// TwinCAT 3 PLC project TcoInspectorsTests
// Title: TcoInspectorsTests
// Company: Vortex.Library
// ProjectVersion: 0.6.0.913
// ProgramVersion: 3.1.4024.12
// libraries:
//   Tc2_Standard, * (Beckhoff Automation GmbH)
//   Tc2_System, * (Beckhoff Automation GmbH)
//   Tc3_Module, * (Beckhoff Automation GmbH)
//   TcoCore, 0.6.0.913 (Vortex.Library)
//   TcoInspectors, 0.6.0.913 (Vortex.Library)
// project tree:
//   GVLs/ GVL.TcGVL
//   / PlcTask.TcTTO
//   POUs/Examples/ ExampleComponents.TcDUT, ExampleContext.TcPOU, ExampleDimensionsInspectors.TcDUT, ExampleInspectorsStruct.TcDUT, Examples_2.TcPOU, ExamplesImplementationWithDone.TcPOU, Sequence1Task.TcPOU
//   POUs/ MAIN.TcPOU
//   POUs/Mocks/ MockCoordinator.TcPOU
//   POUs/Tests/TcoAnalogueInspector/ TcoAnalogueInspectorTests.TcPOU
//   POUs/Tests/TcoDataInspector/ TcoDataInspectorTests.TcPOU
//   POUs/Tests/TcoDigitalInspector/Legacy/ eDigitalInspectorTests.TcDUT, LegacyTcoDigitalInspectorTests.TcPOU
//   POUs/Tests/TcoDigitalInspector/ TcoDigitalInspectorTests.TcPOU
//   POUs/Tests/TcoInspectionGroup/ eInspectionGroupTests.TcDUT, TcoInspectionGroupTests.TcPOU
//   POUs/Tests/TcoInspector/ eInspectorTests.TcDUT, TcoInspectorTests.TcPOU
// (motion and I/O tree: see PLC project tcoinspectors)
// real-time tasks:
//   TASK PlcTask: cycle T#10ms, priority 20, ADS port 350
//   TASK PlcTask1: cycle T#10ms, priority 21, ADS port 351

CONFIGURATION TcoInspectorsTests
    RESOURCE PLC ON TwinCAT3
        TASK PlcTask(INTERVAL := T#10ms, PRIORITY := 21);
        PROGRAM MAIN WITH PlcTask : MAIN;
    END_RESOURCE
END_CONFIGURATION

// ---- POUs/Examples/ExampleComponents.TcDUT
TYPE ExampleComponents EXTENDS TcoCore.TcoStruct :
STRUCT
    DmcReader : STRING;
    BoltPresenceSensor : BOOL;
    DimX_Sensor : LREAL;
    DimY_Sensor : LREAL;
    DimZ_Sensor : LREAL;
END_STRUCT
END_TYPE

// ---- POUs/Examples/ExampleDimensionsInspectors.TcDUT
TYPE ExampleDimensionsInspectors EXTENDS TcoCore.TcoStruct :
STRUCT
    {attribute addProperty Name "Dimension X inspection"}
    DimX_Inspector : TcoInspectors.TcoAnalogueInspector(THISSTRUCT);
    {attribute addProperty Name "Dimension Y inspection"}
    DimY_Inspector : TcoInspectors.TcoAnalogueInspector(THISSTRUCT);
    {attribute addProperty Name "Dimension ZZ inspection"}
    DimZ_Inspector : TcoInspectors.TcoAnalogueInspector(THISSTRUCT);
    {attribute addProperty Name "Dimension Z inspection name is TOOOOOOOO LONG"}
    DimCustom_Inspector : TcoInspectors.TcoAnalogueInspector(THISSTRUCT);
    {attribute addProperty Name "Dimension inspection 1"}
    Dim_Inspector_1 : TcoInspectors.TcoAnalogueInspector(THISSTRUCT);
    {attribute addProperty Name "Dimension inspection 2"}
    Dim_Inspector_2 : TcoInspectors.TcoAnalogueInspector(THISSTRUCT);
    {attribute addProperty Name "Dimension inspection 3"}
    Dim_Inspector_3 : TcoInspectors.TcoAnalogueInspector(THISSTRUCT);
    {attribute addProperty Name "Dimension inspection 4"}
    Dim_Inspector_4 : TcoInspectors.TcoAnalogueInspector(THISSTRUCT);
    {attribute addProperty Name "Dimension inspection 5"}
    Dim_Inspector_5 : TcoInspectors.TcoAnalogueInspector(THISSTRUCT);
    {attribute addProperty Name "Dimension inspection 6"}
    Dim_Inspector_6 : TcoInspectors.TcoAnalogueInspector(THISSTRUCT);
    {attribute addProperty Name "Dimension inspection 7"}
    Dim_Inspector_7 : TcoInspectors.TcoAnalogueInspector(THISSTRUCT);
    {attribute addProperty Name "Dimension inspection 8"}
    Dim_Inspector_8 : TcoInspectors.TcoAnalogueInspector(THISSTRUCT);
    {attribute addProperty Name "Dimension inspection 9"}
    Dim_Inspector_9 : TcoInspectors.TcoAnalogueInspector(THISSTRUCT);
    {attribute addProperty Name "Dimension inspection 10"}
    Dim_Inspector_10 : TcoInspectors.TcoAnalogueInspector(THISSTRUCT);
    {attribute addProperty Name "Dimension inspection 11"}
    Dim_Inspector_11 : TcoInspectors.TcoAnalogueInspector(THISSTRUCT);
    {attribute addProperty Name "Dimension inspection 12"}
    Dim_Inspector_12 : TcoInspectors.TcoAnalogueInspector(THISSTRUCT);
    {attribute addProperty Name "Dimension inspection 13"}
    Dim_Inspector_13 : TcoInspectors.TcoAnalogueInspector(THISSTRUCT);
    {attribute addProperty Name "Dimension inspection 14"}
    Dim_Inspector_14 : TcoInspectors.TcoAnalogueInspector(THISSTRUCT);
    {attribute addProperty Name "Dimension inspection 15"}
    Dim_Inspector_15 : TcoInspectors.TcoAnalogueInspector(THISSTRUCT);
    {attribute addProperty Name "Dimension inspection 16"}
    Dim_Inspector_16 : TcoInspectors.TcoAnalogueInspector(THISSTRUCT);
    {attribute addProperty Name "Dimension inspection 17"}
    Dim_Inspector_17 : TcoInspectors.TcoAnalogueInspector(THISSTRUCT);
    {attribute addProperty Name "Dimension inspection 18"}
    Dim_Inspector_18 : TcoInspectors.TcoAnalogueInspector(THISSTRUCT);
    {attribute addProperty Name "Dimension inspection 19"}
    Dim_Inspector_19 : TcoInspectors.TcoAnalogueInspector(THISSTRUCT);
    {attribute addProperty Name "Dimension inspection 20"}
    Dim_Inspector_20 : TcoInspectors.TcoAnalogueInspector(THISSTRUCT);
//Inspectors : ARRAY[0..20] OF TcoInspectors.TcoAnalogueInspector(THISSTRUCT);
END_STRUCT
END_TYPE

// ---- POUs/Examples/ExampleInspectorsStruct.TcDUT
TYPE ExampleInspectorsStruct EXTENDS TcoCore.TcoStruct :
STRUCT
    {attribute addProperty Name "Overall result"}
    OverallResult : TcoInspectors.TcoComprehensiveResult;
    {attribute addProperty Name "DMC code inspection"}
    DmcInspector : TcoInspectors.TcoDataInspector(THISSTRUCT);
    {attribute addProperty Name "Bolt presence inspection"}
    BoltPresenceInspector : TcoInspectors.TcoDigitalInspector(THISSTRUCT);
    Dimensions : ExampleDimensionsInspectors := (Parent := THISSTRUCT);
END_STRUCT
END_TYPE

// ---- POUs/Tests/TcoDigitalInspector/Legacy/eDigitalInspectorTests.TcDUT
{attribute 'qualified_only'}
{attribute 'strict'}
TYPE eDigitalInspectorTests :
(
    Inspect := 10,
    GetResult := 20,
    UpdateOverall := 30,
    OnFailCarryOn := 40,
    OnFailRetry := 50,
    OnFailTerminate := 60
);
END_TYPE

// ---- POUs/Tests/TcoInspectionGroup/eInspectionGroupTests.TcDUT
{attribute 'qualified_only'}
{attribute 'strict'}
TYPE eInspectionGroupTests :
(
    Inspect := 10,
    GetResult := 20,
    OnFailCarryOn := 40,
    OnFailRetry := 50,
    OnFailTerminate := 60,
    OnFailDiaglog := 70,
    InspectWithNormalizedNumberOfRetries := 80,
    UpdateComprehensiveResultDescriptions := 90
);
END_TYPE

// ---- POUs/Tests/TcoInspector/eInspectorTests.TcDUT
{attribute 'qualified_only'}
{attribute 'strict'}
TYPE eInspectorTests :
(
    Inspect := 10,
    GetResult := 20,
    UpdateOverall := 30,
    OnFailCarryOn := 40,
    OnFailRetry := 50,
    OnFailTerminate := 60,
    OnFailDialog := 70
);
END_TYPE

// ---- GVLs/GVL.TcGVL
{attribute 'qualified_only'}
VAR_GLOBAL
END_VAR

// ---- POUs/MAIN.TcPOU
PROGRAM MAIN
VAR
    _legacyDigitalInspectorTests : LegacyTcoDigitalInspectorTests;
    _digitalInspectorTests : TcoDigitalInspectorTests;
    _analogueInspectorTests : TcoAnalogueInspectorTests;
    _dataInspectorTests : TcoDataInspectorTests;
    _inspectionGroupTests : TcoInspectionGroupTests;
    _exampleContext : ExampleContext;
END_VAR

_legacyDigitalInspectorTests.ProbeRun();
_digitalInspectorTests.ProbeRun();
_analogueInspectorTests.ProbeRun();
_dataInspectorTests.ProbeRun();
_inspectionGroupTests.ProbeRun();
_exampleContext.Run();

END_PROGRAM

// ---- POUs/Tests/TcoDigitalInspector/Legacy/LegacyTcoDigitalInspectorTests.TcPOU
FUNCTION_BLOCK LegacyTcoDigitalInspectorTests EXTENDS TcoCore._internals_TcoContext
VAR
    _sut : TcoInspectors.TcoDigitalInspector(THIS^);
    _inspectedValue : BOOL;
    _result : TcoInspectors.eInspectorResult;
    _isOverIspected : BOOL;
    _overallResult : TcoInspectors.TcoComprehensiveResult;
    _coordinator : MockCoordinator;
    i_coordinator : TcoCore.ITcoCoordinator;
    _retryState : INT;
END_VAR

METHOD PROTECTED Main
i_coordinator := _coordinator;

CASE _testId OF
    0:
        _result := 0;
        _isOverIspected := FALSE;
    eDigitalInspectorTests.Inspect:
        THIS^.ProbeDoneWhen(_sut.Inspect(_inspectedValue).UpdateComprehensiveResult(_overallResult).Done);
    eDigitalInspectorTests.GetResult:
        _result := _sut.Inspect(_inspectedValue).Result;
        _isOverIspected := _sut.Inspect(_inspectedValue).OverInspected;
    eDigitalInspectorTests.OnFailCarryOn:
        THIS^.ProbeDoneWhen(_sut.WithCoordinator(i_coordinator).Inspect(_inspectedValue).OnFail().CarryOn());
    eDigitalInspectorTests.OnFailRetry:
        THIS^.ProbeDoneWhen(_sut.WithCoordinator(i_coordinator).Inspect(_inspectedValue).OnFail().Retry(_retryState));
    eDigitalInspectorTests.OnFailTerminate:
        THIS^.ProbeDoneWhen(_sut.WithCoordinator(i_coordinator).Inspect(_inspectedValue).OnFail().Terminate());
END_CASE
END_METHOD

END_FUNCTION_BLOCK

// ---- POUs/Mocks/MockCoordinator.TcPOU
FUNCTION_BLOCK MockCoordinator IMPLEMENTS TcoCore.ITcoCoordinator
VAR
    _state : INT;
END_VAR

PROPERTY IsFreshState : BOOL
GET
END_GET
END_PROPERTY

METHOD MoveNext : BOOL
_state := _state + 1;
END_METHOD

METHOD Retry : BOOL
VAR_INPUT
    inFromState : INT;
END_VAR
_state := inFromState;
END_METHOD

METHOD Terminate : BOOL
_state := 8005;
END_METHOD

END_FUNCTION_BLOCK

// ---- POUs/Tests/TcoDigitalInspector/TcoDigitalInspectorTests.TcPOU
FUNCTION_BLOCK TcoDigitalInspectorTests EXTENDS TcoInspectorTests
VAR
    _sut : TcoInspectors.TcoDigitalInspector(THIS^);
    _inspectedValue : BOOL;
END_VAR

METHOD Inspect : TcoInspectors.IInspector
Inspect := _sut.Inspect(_inspectedValue);
END_METHOD

METHOD PROTECTED Main
SUPER^.Main();
END_METHOD

METHOD WithCoordinator : REFERENCE TO TcoInspectorTests
VAR_INPUT
    inoCoordinator : TcoCore.ITcoCoordinator;
END_VAR
_sut.WithCoordinator(_coordinator);
WithCoordinator REF= THIS^;
END_METHOD

END_FUNCTION_BLOCK

// ---- POUs/Tests/TcoInspector/TcoInspectorTests.TcPOU
FUNCTION_BLOCK ABSTRACT TcoInspectorTests EXTENDS TcoCore._internals_TcoContext
VAR
    _result : TcoInspectors.eInspectorResult;
    _isOverIspected : BOOL;
    _overallResult : TcoInspectors.TcoComprehensiveResult;
    _coordinator : MockCoordinator;
    i_coordinator : TcoCore.ITcoCoordinator;
    _retryState : INT;
END_VAR

METHOD ABSTRACT Inspect : TcoInspectors.IInspector
END_METHOD

METHOD PROTECTED Main
i_coordinator := _coordinator;

CASE _testId OF
    0:
        _result := 0;
        _isOverIspected := FALSE;
    eInspectorTests.Inspect:
        THIS^.ProbeDoneWhen(Inspect().UpdateComprehensiveResult(_overallResult).Done);
    eInspectorTests.GetResult:
        _result := Inspect().Result;
        _isOverIspected := Inspect().OverInspected;
    eInspectorTests.OnFailCarryOn:
        THIS^.ProbeDoneWhen(WithCoordinator(inoCoordinator := i_coordinator).Inspect().OnFail().CarryOn());
    eInspectorTests.OnFailRetry:
        THIS^.ProbeDoneWhen(WithCoordinator(inoCoordinator := i_coordinator).Inspect().OnFail().Retry(_retryState));
    eInspectorTests.OnFailTerminate:
        THIS^.ProbeDoneWhen(WithCoordinator(inoCoordinator := i_coordinator).Inspect().OnFail().Terminate());
    eInspectorTests.OnFailDialog:
        THIS^.ProbeDoneWhen(WithCoordinator(inoCoordinator := i_coordinator).Inspect().OnFail().Dialog(100));
END_CASE
END_METHOD

METHOD ABSTRACT WithCoordinator : REFERENCE TO TcoInspectorTests
VAR_INPUT
    inoCoordinator : TcoCore.ITcoCoordinator;
END_VAR
END_METHOD

END_FUNCTION_BLOCK

// ---- POUs/Tests/TcoAnalogueInspector/TcoAnalogueInspectorTests.TcPOU
FUNCTION_BLOCK TcoAnalogueInspectorTests EXTENDS TcoInspectorTests
VAR
    _sut : TcoInspectors.TcoAnalogueInspector(THIS^);
    _inspectedValue : LREAL;
END_VAR

METHOD Inspect : TcoInspectors.IInspector
Inspect := _sut.Inspect(_inspectedValue);
END_METHOD

METHOD PROTECTED Main
SUPER^.Main();
END_METHOD

METHOD WithCoordinator : REFERENCE TO TcoInspectorTests
VAR_INPUT
    inoCoordinator : TcoCore.ITcoCoordinator;
END_VAR
_sut.WithCoordinator(_coordinator);
WithCoordinator REF= THIS^;
END_METHOD

END_FUNCTION_BLOCK

// ---- POUs/Tests/TcoDataInspector/TcoDataInspectorTests.TcPOU
FUNCTION_BLOCK TcoDataInspectorTests EXTENDS TcoInspectorTests
VAR
    _sut : TcoInspectors.TcoDataInspector(THIS^);
    _inspectedValue : STRING;
END_VAR

METHOD Inspect : TcoInspectors.IInspector
Inspect := _sut.Inspect(_inspectedValue);
END_METHOD

METHOD PROTECTED Main
SUPER^.Main();
END_METHOD

METHOD WithCoordinator : REFERENCE TO TcoInspectorTests
VAR_INPUT
    inoCoordinator : TcoCore.ITcoCoordinator;
END_VAR
_sut.WithCoordinator(_coordinator);
WithCoordinator REF= THIS^;
END_METHOD

END_FUNCTION_BLOCK

// ---- POUs/Tests/TcoInspectionGroup/TcoInspectionGroupTests.TcPOU
FUNCTION_BLOCK TcoInspectionGroupTests EXTENDS TcoCore._internals_TcoContext
VAR
    _sut : TcoInspectors.TcoInspectionGroup(THIS^);
    _diis : ARRAY[0..1] OF TcoInspectors.TcoDigitalInspector(THIS^);
    _dii_inspectedValues : ARRAY[0..1] OF BOOL;
    _dais : ARRAY[0..1] OF TcoInspectors.TcoAnalogueInspector(THIS^);
    _dai_inspectedValues : ARRAY[0..1] OF REAL;
    _ddis : ARRAY[0..1] OF TcoInspectors.TcoDataInspector(THIS^);
    _ddi_inspectedValues : ARRAY[0..1] OF STRING;
    _overallResult : TcoInspectors.TcoComprehensiveResult;
    _coordinator : MockCoordinator;
    _retryState : INT;
    _tmp : ITcoInspectionGroupAct;
END_VAR

METHOD PROTECTED Main
CASE _testId OF
    eInspectionGroupTests.Inspect:
        THIS^.ProbeDoneWhen(_sut.Act()
                .Inspect(_diis[0].Inspect(_dii_inspectedValues[0]))
                .Inspect(_diis[1].Inspect(_dii_inspectedValues[1]))
                .Inspect(_dais[0].Inspect(_dai_inspectedValues[0]))
                .Inspect(_dais[1].Inspect(_dai_inspectedValues[1]))
                .Inspect(_ddis[0].Inspect(_ddi_inspectedValues[0]))
                .Inspect(_ddis[1].Inspect(_ddi_inspectedValues[1]))
                .UpdateComprehensiveResult(_overallResult).Done);
    eInspectionGroupTests.OnFailCarryOn:
        THIS^.ProbeDoneWhen(_sut.WithCoordinator(_coordinator)
                .Act()
                .Inspect(_diis[0].Inspect(_dii_inspectedValues[0]))
                .Inspect(_diis[1].Inspect(_dii_inspectedValues[1]))
                .Inspect(_dais[0].Inspect(_dai_inspectedValues[0]))
                .Inspect(_dais[1].Inspect(_dai_inspectedValues[1]))
                .Inspect(_ddis[0].Inspect(_ddi_inspectedValues[0]))
                .Inspect(_ddis[1].Inspect(_ddi_inspectedValues[1]))
                .UpdateComprehensiveResult(_overallResult)
                .OnFail()
                .CarryOn());
    eInspectionGroupTests.OnFailRetry:
        THIS^.ProbeDoneWhen(_sut.WithCoordinator(_coordinator)
                .Act()
                .Inspect(_diis[0].Inspect(_dii_inspectedValues[0]))
                .Inspect(_diis[1].Inspect(_dii_inspectedValues[1]))
                .Inspect(_dais[0].Inspect(_dai_inspectedValues[0]))
                .Inspect(_dais[1].Inspect(_dai_inspectedValues[1]))
                .Inspect(_ddis[0].Inspect(_ddi_inspectedValues[0]))
                .Inspect(_ddis[1].Inspect(_ddi_inspectedValues[1]))
                .UpdateComprehensiveResult(_overallResult)
                .OnFail()
                .Retry(_retryState));
    eInspectionGroupTests.OnFailTerminate:
        THIS^.ProbeDoneWhen(_sut.WithCoordinator(_coordinator)
                .Act()
                .Inspect(_diis[0].Inspect(_dii_inspectedValues[0]))
                .Inspect(_diis[1].Inspect(_dii_inspectedValues[1]))
                .Inspect(_dais[0].Inspect(_dai_inspectedValues[0]))
                .Inspect(_dais[1].Inspect(_dai_inspectedValues[1]))
                .Inspect(_ddis[0].Inspect(_ddi_inspectedValues[0]))
                .Inspect(_ddis[1].Inspect(_ddi_inspectedValues[1]))
                .UpdateComprehensiveResult(_overallResult)
                .OnFail()
                .Terminate());
    eInspectionGroupTests.OnFailDiaglog:
        THIS^.ProbeDoneWhen(_sut.WithCoordinator(_coordinator)
                .Act()
                .Inspect(_diis[0].Inspect(_dii_inspectedValues[0]))
                .Inspect(_diis[1].Inspect(_dii_inspectedValues[1]))
                .Inspect(_dais[0].Inspect(_dai_inspectedValues[0]))
                .Inspect(_dais[1].Inspect(_dai_inspectedValues[1]))
                .Inspect(_ddis[0].Inspect(_ddi_inspectedValues[0]))
                .Inspect(_ddis[1].Inspect(_ddi_inspectedValues[1]))
                .UpdateComprehensiveResult(_overallResult)
                .OnFail()
                .Dialog(100));
    eInspectionGroupTests.InspectWithNormalizedNumberOfRetries:
        THIS^.ProbeDoneWhen(_sut.WithCoordinator(_coordinator)
                .Act()
                .NormalizeRetries(_diis[0])
                .NormalizeRetries(_diis[1])
                .NormalizeRetries(_dais[0])
                .NormalizeRetries(_dais[1])
                .NormalizeRetries(_ddis[0])
                .NormalizeRetries(_ddis[1])
                .Inspect(_diis[0].Inspect(_dii_inspectedValues[0]))
                .Inspect(_diis[1].Inspect(_dii_inspectedValues[1]))
                .Inspect(_dais[0].Inspect(_dai_inspectedValues[0]))
                .Inspect(_dais[1].Inspect(_dai_inspectedValues[1]))
                .Inspect(_ddis[0].Inspect(_ddi_inspectedValues[0]))
                .Inspect(_ddis[1].Inspect(_ddi_inspectedValues[1]))
                .UpdateComprehensiveResult(_overallResult).Done);
    eInspectionGroupTests.UpdateComprehensiveResultDescriptions:
        THIS^.ProbeDoneWhen(_sut.WithCoordinator(_coordinator)
                .Act()
                .NormalizeRetries(_diis[0])
                .NormalizeRetries(_diis[1])
                .NormalizeRetries(_dais[0])
                .NormalizeRetries(_dais[1])
                .NormalizeRetries(_ddis[0])
                .NormalizeRetries(_ddis[1])
                .Inspect(_diis[0].Inspect(_dii_inspectedValues[0]))
                .Inspect(_diis[1].Inspect(_dii_inspectedValues[1]))
                .Inspect(_dais[0].Inspect(_dai_inspectedValues[0]))
                .Inspect(_dais[1].Inspect(_dai_inspectedValues[1]))
                .Inspect(_ddis[0].Inspect(_ddi_inspectedValues[0]))
                .Inspect(_ddis[1].Inspect(_ddi_inspectedValues[1]))
                .UpdateComprehensiveResult(_overallResult)
                .OnFail()
                .Dialog(100));
END_CASE
END_METHOD

END_FUNCTION_BLOCK

// ---- POUs/Examples/ExampleContext.TcPOU
FUNCTION_BLOCK ExampleContext EXTENDS TcoCore.TcoContext
VAR
    Data            : ExampleInspectorsStruct := (Parent := THIS^);
    Components      : ExampleComponents       := (Parent := THIS^);
    GroupInspection : TcoInspectors.TcoInspectionGroup(THIS^);
    _sequence1      : TcoCore.TcoSequence(THIS^, eRestoreMode.None);
    _observer       : TcoCore.TcoSequencerObserver(THIS^);
    {attribute addProperty Name "Start sequence"}
    _sequence1Task 	: Sequence1Task(THIS^);
    _dialog        	: TcoCore.TcoDialog(THIS^);
    {attribute 'hide'}
    EmptyData 		: ExampleInspectorsStruct := (Parent := THIS^);

    _examples_2 	: Examples_2(THIS^);
	_examplesImplementationWithDone : ExamplesImplementationWithDone(THIS^);
	_tonRetry: TON;
	_rtrigRetry: R_trig;
	_tonTerminate: TON;
	testRetry:BOOL;
	testTerminate:BOOL;
	
END_VAR

(*~
	<docu>
		<summary>
			Main method of the TcoContext. This is the entry point of any control logic that belongs to this context. 
			The call of this method is ensured by calling the <c>InstanceName.Run()</c> method, and it must not be called explicitly.
			This method is abstract, and it must be overridden in derived block.
		</summary>
	</docu>
~*)
METHOD PROTECTED  Main
_sequence1Task(Sequence := _sequence1);
IF(_sequence1Task.Execute())THEN
	Sequence1();
END_IF;

_examples_2();
_examplesImplementationWithDone();
END_METHOD

METHOD Sequence1
VAR
    seq    : REFERENCE TO TcoCore.TcoSequence;
    answer : TcoCore.eDialogAnswer;
	i: INT;
END_VAR
seq REF= _sequence1;

seq.Open();
seq.Observer := _observer;

IF (seq.Step(inStepID := 0,
    inEnabled := TRUE,
    inStepDescription := 'ASKING SOME QUESTION')) THEN
    //--------------------------------------------------------
    //<StandardDialog>	
    //restore method also close inactive dialog
    Data.BoltPresenceInspector.Restore();
    GroupInspection.Restore();
    SetupData();
    answer := _dialog
        .Show()
        .WithType(eDialogType.Question)
        .WithCaption('Ready to go?')
        .WithText('We are about to start the inspection sequence. Do we go ahead?')
        .WithYesNoCancel().Answer;

    //

    IF (answer = TcoCore.eDialogAnswer.Yes) THEN
        seq.CompleteStep();
    ELSIF (answer = TcoCore.eDialogAnswer.No) THEN
        _sequence1Task.Restore();
    ELSIF (answer = TcoCore.eDialogAnswer.Cancel) THEN
        seq.RequestStep(400);
    END_IF;
    //</StandardDialog>	 
    //--------------------------------------------------------			
END_IF;

IF (seq.Step(inStepID := 25,
    inEnabled := TRUE,
    inStepDescription := 'SETUP DATA')) THEN
    //--------------------------------------------------------    
    SetupData();
    seq.CompleteStep();
    //--------------------------------------------------------			
END_IF;

IF (seq.Step(inStepID := 50,
    inEnabled := TRUE,
    inStepDescription := 'INIT')) THEN
    //--------------------------------------------------------    	 	       
    seq.CompleteStep();
    //--------------------------------------------------------			
END_IF;

IF (seq.Step(inStepID := 100,
    inEnabled := TRUE,
    inStepDescription := 'INSPECT DMC CODE - WHEN CARRY ON')) THEN
    //--------------------------------------------------------
    Data.DmcInspector.WithCoordinator(seq)
        .Inspect(Components.DmcReader)
        .UpdateComprehensiveResult(Data.OverallResult)
        .OnFail()
        .CarryOn();
    //--------------------------------------------------------			
END_IF;

IF (seq.Step(inStepID := 105,
    inEnabled := TRUE,
    inStepDescription := 'SETUP DATA')) THEN
    //--------------------------------------------------------    
    SetupData();
    seq.CompleteStep();
    //--------------------------------------------------------			
END_IF;

IF (seq.Step(inStepID := 110,
    inEnabled := TRUE,
    inStepDescription := 'DUMMY WAIT')) THEN
    //--------------------------------------------------------
    seq.StepCompleteWhen(Seq.CurrentStep.Duration > T#1S);
    //--------------------------------------------------------			
END_IF;

IF (seq.Step(inStepID := 120,
    inEnabled := TRUE,
    inStepDescription := 'INSPECT DMC CODE -  RETRY THEN TERMINATE')) THEN
    //--------------------------------------------------------
    Data.DmcInspector.WithCoordinator(seq)
        .Inspect(Components.DmcReader)
        .UpdateComprehensiveResult(Data.OverallResult)
        .OnFail()
        .RetryThenTerminate(110);
    //--------------------------------------------------------			
END_IF;

//<TcoDigitalInspector>	
IF (seq.Step(inStepID := 200,
    inEnabled := true,
    inStepDescription := 'INSPECT BOLT PRESENCE - ASK WHAT TO DO')) THEN
    //--------------------------------------------------------	
    IF seq.IsFreshState THEN
        SetupData();
    END_IF

    Data.BoltPresenceInspector
        .WithCoordinator(seq)
        .Inspect(Components.BoltPresenceSensor)
        .UpdateComprehensiveResult(Data.OverallResult)
        .OnFail()
        .Dialog(seq.CurrentStep.ID + 1);
    //--------------------------------------------------------			
END_IF;

IF (seq.Step(inStepID := 201,
    inEnabled := true,
    inStepDescription := 'INSPECT BOLT PRESENCE - ASK WHAT TO DO WITH INSTRUCTION')) THEN
    //--------------------------------------------------------	
    IF seq.IsFreshState THEN
        SetupData();
    END_IF

    Data.BoltPresenceInspector
        .WithCoordinator(seq)
        .Inspect(Components.BoltPresenceSensor)
        .UpdateComprehensiveResult(Data.OverallResult)
        .Instruct('Something is wrong')
        .OnFail()
        .Dialog(seq.CurrentStep.ID + 1);
    //--------------------------------------------------------			
END_IF;

IF (seq.Step(inStepID := 202,
    inEnabled := true,
    inStepDescription := 'INSPECT BOLT PRESENCE - ASK WHAT TO DO WITH INSTRUCTION AND PICTURE')) THEN
    //--------------------------------------------------------	
    IF seq.IsFreshState THEN
        SetupData();
    END_IF

    Data.BoltPresenceInspector
        .WithCoordinator(seq)
        .Inspect(Components.BoltPresenceSensor)
        .UpdateComprehensiveResult(Data.OverallResult)
        .Instruct('Something is wrong')
        .InstructWithImage('d:\MTS\Develop\TcOpenGroup\TcOpen\assets\logo\TcOpenWide.png', 200, 200)
        .OnFail()
        .Dialog(seq.CurrentStep.ID + 1);
    //--------------------------------------------------------			
END_IF;

IF (seq.Step(inStepID := 203,
    inEnabled := true,
    inStepDescription := 'INSPECT BOLT PRESENCE - ASK WHAT TO DO WITH INSTRUCTION AND BIGGER PICTURE')) THEN
    //--------------------------------------------------------	
    IF seq.IsFreshState THEN
        SetupData();
    END_IF

    Data.BoltPresenceInspector
        .WithCoordinator(seq)
        .Inspect(Components.BoltPresenceSensor)
        .UpdateComprehensiveResult(Data.OverallResult)
        .Instruct('Something is wrong') //provide cuastomized instruction instead of automaticaly generated
        .InstructWithImage('d:\MTS\Develop\TcOpenGroup\TcOpen\assets\logo\TcOpenWide.png', 600, 600)
        .OnFail()
        .Dialog(seq.CurrentStep.ID + 1);
    //--------------------------------------------------------			
END_IF;

IF (seq.Step(inStepID := 204,
    inEnabled := true,
    inStepDescription := 'INSPECT BOLT PRESENCE - ASK WHAT TO DO WITH FAILURE DESCRIPTION')) THEN
    //--------------------------------------------------------	
    IF seq.IsFreshState THEN
        SetupData();
    END_IF

    Data.BoltPresenceInspector
        .WithCoordinator(seq)
        .Inspect(Components.BoltPresenceSensor)
        .UpdateComprehensiveResult(Data.OverallResult)
        .WithFailureDescription()
        .OnFail()
        .Dialog(seq.CurrentStep.ID + 1);
    //--------------------------------------------------------			
END_IF;

IF (seq.Step(inStepID := 205,
    inEnabled := true,
    inStepDescription := 'INSPECT BOLT PRESENCE - ASK WHAT TO DO WITH DESCRIPTION')) THEN
    //--------------------------------------------------------	
    IF seq.IsFreshState THEN
        SetupData();
    END_IF

    Data.BoltPresenceInspector
        .WithCoordinator(seq)
        .Inspect(Components.BoltPresenceSensor)
        .UpdateComprehensiveResult(Data.OverallResult)
        .WithDescription() //provide description of Inspector in this case will be Bolt presence inspection because...	{attribute addProperty Name "Bolt presence inspection"}
        .OnFail()
        .Dialog(seq.CurrentStep.ID + 1);
    //--------------------------------------------------------			
END_IF;

IF (seq.Step(inStepID := 206,
    inEnabled := true,
    inStepDescription := 'INSPECT BOLT PRESENCE - ASK WHAT TO DO WITH FAILURE DESCRIPTION AND ERROR CODE(IF DEFINED)')) THEN
    //--------------------------------------------------------	
    IF seq.IsFreshState THEN
        SetupData();
    END_IF

    Data.BoltPresenceInspector
        .WithCoordinator(seq)
        .Inspect(Components.BoltPresenceSensor)
        .UpdateComprehensiveResult(Data.OverallResult)
        .WithErrorCode()
        .WithFailureDescription()
        .OnFail()
        .Dialog(250);
    //--------------------------------------------------------			
END_IF;

IF (seq.Step(inStepID := 250,
    inEnabled := TRUE,
    inStepDescription := 'INSPECT BOLT PRESENCE - ASK WHAT TO DO WITH EXTERNAL CLOSE')) THEN
    //--------------------------------------------------------	
    IF seq.IsFreshState THEN
        SetupData();
    END_IF

    Data.BoltPresenceInspector
        .WithCoordinator(seq)
        .Inspect(Components.BoltPresenceSensor)
        .UpdateComprehensiveResult(Data.OverallResult)
        .OnFail()
        .DialogWithExternalClose(250, inRetrySignal := testRetry, inTerminateSignal := testTerminate);
    //--------------------------------------------------------			
END_IF;

IF (seq.Step(inStepID := 300,
    inEnabled := TRUE,
    inStepDescription := 'INSPECT DIMENSIONS - WITH NORMALIZE RETRIES (lower `number of allowed retries` for this call of inspection group)')) THEN
    //--------------------------------------------------------
    IF seq.IsFreshState THEN
        SetupData();
    END_IF

    GroupInspection
        .WithCoordinator(seq)
        .Act()
        .NormalizeRetries(Data.Dimensions.DimX_Inspector)
        .NormalizeRetries(Data.Dimensions.DimY_Inspector)
        .NormalizeRetries(Data.Dimensions.DimZ_Inspector)
        .Inspect(Data.Dimensions.DimX_Inspector.Inspect(Components.DimX_Sensor))
        .Inspect(Data.Dimensions.DimY_Inspector.Inspect(Components.DimY_Sensor))
        .Inspect(Data.Dimensions.DimZ_Inspector.Inspect(Components.DimZ_Sensor))
        .UpdateComprehensiveResult(Data.OverallResult)
        .OnFail()
        .Dialog(300);
    //--------------------------------------------------------			
END_IF;

IF (seq.Step(inStepID := 309,
    inEnabled := TRUE,
    inStepDescription := 'INSPECT MULTI DIMENSIONS - EXTERNAL CLOSE')) THEN
    //--------------------------------------------------------
    IF seq.IsFreshState THEN
        SetupData();
    END_IF

    GroupInspection
        .WithCoordinator(seq)
        .Act();

    GroupInspection.Inspect(Data.Dimensions.DimX_Inspector.Inspect(Components.DimX_Sensor));
    GroupInspection.Inspect(Data.Dimensions.DimY_Inspector.WithCoordinator(seq).Inspect(Components.DimY_Sensor));
    GroupInspection.Inspect(Data.Dimensions.DimZ_Inspector.WithCoordinator(seq).Inspect(Components.DimZ_Sensor));

    GroupInspection.UpdateComprehensiveResult(Data.OverallResult)
        .Instruct('Something is wrong')
        .InstructWithImage('d:\MTS\Develop\TcOpenGroup\TcOpen\assets\logo\TcOpenWide.png', 400, 600)
        .HideTerminate()
        .OnFail()
        .DialogWithExternalClose(309, inRetrySignal := testRetry, inTerminateSignal := testTerminate);

    //--------------------------------------------------------			
END_IF

IF (seq.Step(inStepID := 310,
    inEnabled := TRUE,
    inStepDescription := 'INSPECT MULTI DIMENSIONS - EXTERNAL CLOSE')) THEN
    //--------------------------------------------------------
    IF seq.IsFreshState THEN
        SetupData();
    END_IF

    GroupInspection
        .WithCoordinator(seq)
        .Act();

    GroupInspection.Inspect(Data.Dimensions.Dim_Inspector_1.WithCoordinator(seq).Inspect(Components.DimZ_Sensor));
    GroupInspection.Inspect(Data.Dimensions.Dim_Inspector_2.WithCoordinator(seq).Inspect(Components.DimZ_Sensor));
    GroupInspection.Inspect(Data.Dimensions.Dim_Inspector_3.WithCoordinator(seq).Inspect(Components.DimZ_Sensor));
    GroupInspection.Inspect(Data.Dimensions.Dim_Inspector_4.WithCoordinator(seq).Inspect(Components.DimZ_Sensor));
    GroupInspection.Inspect(Data.Dimensions.Dim_Inspector_5.WithCoordinator(seq).Inspect(Components.DimZ_Sensor));
    GroupInspection.Inspect(Data.Dimensions.Dim_Inspector_6.WithCoordinator(seq).Inspect(Components.DimZ_Sensor));
    GroupInspection.Inspect(Data.Dimensions.Dim_Inspector_7.WithCoordinator(seq).Inspect(1));
    GroupInspection.Inspect(Data.Dimensions.Dim_Inspector_8.WithCoordinator(seq).Inspect(Components.DimZ_Sensor));
    GroupInspection.Inspect(Data.Dimensions.Dim_Inspector_9.WithCoordinator(seq).Inspect(Components.DimZ_Sensor));
    GroupInspection.Inspect(Data.Dimensions.Dim_Inspector_10.WithCoordinator(seq).Inspect(Components.DimZ_Sensor));

    GroupInspection.UpdateComprehensiveResult(Data.OverallResult)
        .Instruct('Something is wrong')
        .InstructWithImage('d:\MTS\Develop\TcOpenGroup\TcOpen\assets\logo\TcOpenWide.png', 400, 600)
        .OnFail()
        .DialogWithExternalClose(311, inRetrySignal := testRetry, inTerminateSignal := testTerminate);

    //--------------------------------------------------------			
END_IF

IF (seq.Step(inStepID := 311,
    inEnabled := TRUE,
    inStepDescription := 'INSPECT MULTI DIMENSIONS - EXTERNAL CLOSE')) THEN
    //--------------------------------------------------------
    IF seq.IsFreshState THEN
        SetupData();
    END_IF

    GroupInspection
        .WithCoordinator(seq)
        .Act();

    GroupInspection.Inspect(Data.Dimensions.Dim_Inspector_11.WithCoordinator(seq).Inspect(Components.DimZ_Sensor));
    GroupInspection.Inspect(Data.Dimensions.Dim_Inspector_12.WithCoordinator(seq).Inspect(Components.DimZ_Sensor));
    GroupInspection.Inspect(Data.Dimensions.Dim_Inspector_13.WithCoordinator(seq).Inspect(Components.DimZ_Sensor));
    GroupInspection.Inspect(Data.Dimensions.Dim_Inspector_14.WithCoordinator(seq).Inspect(Components.DimZ_Sensor));
    GroupInspection.Inspect(Data.Dimensions.Dim_Inspector_15.WithCoordinator(seq).Inspect(Components.DimZ_Sensor));
    GroupInspection.Inspect(Data.Dimensions.Dim_Inspector_16.WithCoordinator(seq).Inspect(Components.DimZ_Sensor));
    GroupInspection.Inspect(Data.Dimensions.Dim_Inspector_17.WithCoordinator(seq).Inspect(1));
    GroupInspection.Inspect(Data.Dimensions.Dim_Inspector_18.WithCoordinator(seq).Inspect(Components.DimZ_Sensor));
    GroupInspection.Inspect(Data.Dimensions.Dim_Inspector_19.WithCoordinator(seq).Inspect(Components.DimZ_Sensor));
    GroupInspection.Inspect(Data.Dimensions.Dim_Inspector_20.WithCoordinator(seq).Inspect(Components.DimZ_Sensor));

    GroupInspection.UpdateComprehensiveResult(Data.OverallResult)
        .Instruct('Something is wrong')
        .InstructWithImage('d:\MTS\Develop\TcOpenGroup\TcOpen\assets\logo\TcOpenWide.png', 400, 600)
        .OnFail()
        .DialogWithExternalClose(312, inRetrySignal := testRetry, inTerminateSignal := testTerminate);

    //--------------------------------------------------------			
END_IF

IF (seq.Step(inStepID := 312,
    inEnabled := TRUE,
    inStepDescription := 'INSPECT MULTI DIMENSIONS - EXTERNAL CLOSE WITH FAILED DESCRIPTION')) THEN
    //--------------------------------------------------------
    IF seq.IsFreshState THEN
        SetupData();
    END_IF

    GroupInspection
        .WithCoordinator(seq)
        .Act();

    GroupInspection.Inspect(Data.Dimensions.DimX_Inspector.Inspect(Components.DimX_Sensor));
    GroupInspection.Inspect(Data.Dimensions.DimY_Inspector.WithCoordinator(seq).Inspect(10));
    GroupInspection.Inspect(Data.Dimensions.DimZ_Inspector.WithCoordinator(seq).Inspect(Components.DimZ_Sensor));

    GroupInspection.UpdateComprehensiveResult(Data.OverallResult)
        .Instruct('Something is wrong tooooooooooooooooooo  loooooooooooooooooooooooooooooooooooooooooooooooong')
        .InstructWithImage('d:\MTS\Develop\TcOpenGroup\TcOpen\assets\logo\TcOpenWide.png', 400, 600)
        .WithDescription()
        .OnFail()
        .DialogWithExternalClose(310, inRetrySignal := testRetry, inTerminateSignal := testTerminate);

    //--------------------------------------------------------			
END_IF;

IF (seq.Step(inStepID := 400,
    inEnabled := TRUE,
    inStepDescription := 'DUMMY WAIT')) THEN
    //--------------------------------------------------------

    SetupData();

    seq.StepCompleteWhen(TRUE);
    //--------------------------------------------------------			
END_IF;

IF (seq.Step(inStepID := 405,
    inEnabled := TRUE,
    inStepDescription := 'DUMMY WAIT')) THEN
    //--------------------------------------------------------

    seq.StepCompleteWhen(Seq.CurrentStep.Duration > T#1S);
    //--------------------------------------------------------			
END_IF;

IF (seq.Step(inStepID := 410,
    inEnabled := TRUE,
    inStepDescription := 'INSPECT BOLT PRESENCE - WITH EVALUATE')) THEN
    //--------------------------------------------------------	

    Data.BoltPresenceInspector
        .WithCoordinator(seq)
        .Inspect(Components.BoltPresenceSensor)
        .UpdateComprehensiveResult(Data.OverallResult)
        .OnFail()
        .Evaluate(405, eTcoInspectorFailMode.RetryThenCarryOn, 420);
    //--------------------------------------------------------			
END_IF;

IF (seq.Step(inStepID := 415,
    inEnabled := TRUE,
    inStepDescription := 'DUMMY WAIT')) THEN
    //--------------------------------------------------------

    SetupData();

    seq.StepCompleteWhen(TRUE);
    //--------------------------------------------------------			
END_IF;
IF (seq.Step(inStepID := 416,
    inEnabled := TRUE,
    inStepDescription := 'DUMMY WAIT')) THEN
    //--------------------------------------------------------
    seq.StepCompleteWhen(Seq.CurrentStep.Duration > T#1S);
    //--------------------------------------------------------			
END_IF;


IF (seq.Step(inStepID := 420,
    inEnabled := TRUE,
    inStepDescription := 'INSPECT MULTI DIMENSIONS - WITH EVALUATE')) THEN
    //--------------------------------------------------------

    GroupInspection
        .WithCoordinator(seq)
        .Act();

    GroupInspection.Inspect(Data.Dimensions.DimX_Inspector.Inspect(Components.DimX_Sensor));
    GroupInspection.Inspect(Data.Dimensions.DimY_Inspector.WithCoordinator(seq).Inspect(10));
    GroupInspection.Inspect(Data.Dimensions.DimZ_Inspector.WithCoordinator(seq).Inspect(Components.DimZ_Sensor));

    GroupInspection.UpdateComprehensiveResult(Data.OverallResult)
        .Instruct('Something is wrong tooooooooooooooooooo  loooooooooooooooooooooooooooooooooooooooooooooooong')
        .InstructWithImage('d:\MTS\Develop\TcOpenGroup\TcOpen\assets\logo\TcOpenWide.png', 400, 600)
        .WithDescription()
        .OnFail()
        .Evaluate(415, eTcoInspectorFailMode.JumpTo, 450);

    //--------------------------------------------------------			
END_IF;

IF (seq.Step(inStepID := 450,
    inEnabled := TRUE,
    inStepDescription := 'PREPAIR DATA ')) THEN
    //--------------------------------------------------------

    SetupData();

    seq.StepCompleteWhen(TRUE);
    //--------------------------------------------------------			
END_IF;

IF (seq.Step(inStepID := 451,
    inEnabled := TRUE,
    inStepDescription := 'DUMMY WAIT')) THEN
    //--------------------------------------------------------
    seq.StepCompleteWhen(Seq.CurrentStep.Duration > T#1S);
    //--------------------------------------------------------			
END_IF;


IF (seq.Step(inStepID := 452,
    inEnabled := TRUE,
    inStepDescription := 'INSPECT MULTI DIMENSIONS - WITH EVALUATE RETRY OPTION')) THEN
    //--------------------------------------------------------

    GroupInspection
        .WithCoordinator(seq)
        .Act();

    GroupInspection.Inspect(Data.Dimensions.DimX_Inspector.Inspect(Components.DimX_Sensor));
    GroupInspection.Inspect(Data.Dimensions.DimY_Inspector.Inspect(Components.DimY_Sensor));
    GroupInspection.Inspect(Data.Dimensions.DimZ_Inspector.Inspect(Components.DimZ_Sensor));

    GroupInspection.UpdateComprehensiveResult(Data.OverallResult)
        .Instruct('Something is wrong tooooooooooooooooooo  loooooooooooooooooooooooooooooooooooooooooooooooong')
        .InstructWithImage('d:\MTS\Develop\TcOpenGroup\TcOpen\assets\logo\TcOpenWide.png', 400, 600)
        .WithDescription()
        .OnFail()
        .Evaluate(451, eTcoInspectorFailMode.RetryThenTeminate, 452);

    //--------------------------------------------------------			
END_IF;

IF (seq.Step(inStepID := seq.RESTORE_STEP_ID,
    inEnabled := TRUE,
    inStepDescription := 'RETURN TO THE START OF THE SEQUENCE')) THEN
    //--------------------------------------------------------	
    seq.CompleteSequence();
    //--------------------------------------------------------			
END_IF;

seq.Close();
END_METHOD

METHOD SetupData
VAR_INPUT
END_VAR
//Data := EmptyData;

Data.DmcInspector.Data.RequiredStatus := 'A#*';
Data.DmcInspector.Data.StarNotationEnabled := TRUE;
Data.DmcInspector.Data.PassTime := T#1500MS;
Data.DmcInspector.Data.FailTime := T#2S;
Data.DmcInspector.Data.FailureDescription := 'Data inspection failed';
Data.DmcInspector.Data.ErrorCode := '1';
Data.DmcInspector.Data.RetryAttemptsCount := 0;
Data.DmcInspector.Data.NumberOfAllowedRetries := 5;

Data.BoltPresenceInspector.Data.RequiredStatus := TRUE;
Data.BoltPresenceInspector.Data.PassTime := T#1500MS;
Data.BoltPresenceInspector.Data.FailTime := T#2S;
Data.BoltPresenceInspector.Data.NumberOfAllowedRetries := 2;
Data.BoltPresenceInspector.Data.FailureDescription := 'Bolt inspection failed';
Data.BoltPresenceInspector.Data.ErrorCode := '2';
Data.BoltPresenceInspector.Data.RetryAttemptsCount := 0;

Data.Dimensions.DimX_Inspector.Data.PassTime := T#1500MS;
Data.Dimensions.DimX_Inspector.Data.FailTime := T#2S;
Data.Dimensions.DimX_Inspector.Data.RequiredMin := 9.75;
Data.Dimensions.DimX_Inspector.Data.RequiredMax := 10.25;
Data.Dimensions.DimX_Inspector.Data.NumberOfAllowedRetries := 0;
Data.Dimensions.DimX_Inspector.Data.FailureDescription := 'Dimx inspection failed';
Data.Dimensions.DimX_Inspector.Data.ErrorCode := '3';
Data.Dimensions.DimX_Inspector.Data.RetryAttemptsCount := 0;

Data.Dimensions.DimY_Inspector.Data.PassTime := T#1500MS;
Data.Dimensions.DimY_Inspector.Data.FailTime := T#2S;
Data.Dimensions.DimY_Inspector.Data.RequiredMin := 9.75;
Data.Dimensions.DimY_Inspector.Data.RequiredMax := 10.25;
Data.Dimensions.DimY_Inspector.Data.FailureDescription := 'Dimy inspection failed';
Data.Dimensions.DimY_Inspector.Data.ErrorCode := '4';

Data.Dimensions.DimZ_Inspector.Data.PassTime := T#1500MS;
Data.Dimensions.DimZ_Inspector.Data.FailTime := T#2S;
Data.Dimensions.DimZ_Inspector.Data.RequiredMin := 9.75;
Data.Dimensions.DimZ_Inspector.Data.RequiredMax := 10.25;
Data.Dimensions.DimZ_Inspector.Data.FailureDescription := 'Dimz inspection failed';
Data.Dimensions.DimZ_Inspector.Data.ErrorCode := '5';
END_METHOD

END_FUNCTION_BLOCK

// ---- POUs/Examples/Sequence1Task.TcPOU
FUNCTION_BLOCK Sequence1Task EXTENDS TcoCore.TcoTask
VAR_INPUT
    Sequence : TcoCore.ITcoSequencer;
END_VAR

(*~
    <docu>
        <summary>
            Restores this instance to the Ready state. Can be called explicitly or from within one of the restore mechanisms.
            <para>
                See also <see cref="PlcDocu.TcoCore.TcoTask.AutoRestorable()"/>
            </para>
        </summary>
    </docu>
~*)
METHOD Restore : ITcoRestorable
SUPER^.Restore();
THIS^.Sequence.Restore();
END_METHOD

END_FUNCTION_BLOCK

// ---- POUs/Examples/Examples_2.TcPOU
FUNCTION_BLOCK Examples_2 EXTENDS TcoCore.TcoObject
VAR
    _diSignal : BOOL;
    _di : TcoInspectors.TcoDigitalInspector(THIS^);
    _diTask : TcoCore.TcoTask(THIS^);
    _daSignal : LREAL;
    _da : TcoInspectors.TcoAnalogueInspector(THIS^);
    _daTask : TcoCore.TcoTask(THIS^);
    _ddSignal : STRING;
    _dd : TcoInspectors.TcoDataInspector(THIS^);
    _ddTask : TcoCore.TcoTask(THIS^);
END_VAR

IF (_diTask.Execute()) THEN
    IF (_di.Inspect(_diSignal).Done) THEN
        IF (_di.Result = TcoInspectors.eInspectorResult.Failed) THEN
            _di.Messenger.Build().Append('I failed').As().AsInfo().Pin();
        ELSIF (_di.Result = TcoInspectors.eInspectorResult.Passed) THEN
            _di.Messenger.Build().Append('I passed').As().AsInfo().Pin();
        END_IF
    END_IF;
END_IF;

IF (_daTask.Execute()) THEN
    IF (_da.Inspect(_daSignal).Done) THEN
        IF (_da.Result = TcoInspectors.eInspectorResult.Failed) THEN
            _da.Messenger.Build().Append('I failed').As().AsInfo().Pin();
        ELSIF (_da.Result = TcoInspectors.eInspectorResult.Passed) THEN
            _da.Messenger.Build().Append('I passed').As().AsInfo().Pin();
        END_IF
    END_IF;
END_IF;

IF (_ddTask.Execute()) THEN
    IF (_dd.Inspect(_ddSignal).Done) THEN
        IF (_dd.Result = TcoInspectors.eInspectorResult.Failed) THEN
            _dd.Messenger.Build().Append('I failed').As().AsInfo().Pin();
        ELSIF (_dd.Result = TcoInspectors.eInspectorResult.Passed) THEN
            _dd.Messenger.Build().Append('I passed').As().AsInfo().Pin();
        END_IF
    END_IF;
END_IF;

END_FUNCTION_BLOCK

// ---- POUs/Examples/ExamplesImplementationWithDone.TcPOU
FUNCTION_BLOCK ExamplesImplementationWithDone EXTENDS TcoCore.TcoObject
VAR
    _inspectorsSignal : BOOL;
    _inspector : TcoInspectors.TcoDigitalInspector(THIS^);
    _inspectorTask : TcoCore.TcoTask(THIS^);
END_VAR

IF (_inspectorTask.Execute()) THEN
    IF (_inspector.Inspect(_inspectorsSignal).Done) THEN
        IF (_inspector.Result = TcoInspectors.eInspectorResult.Failed) THEN
            _inspector.Messenger.Build().Append('I failed').As().AsInfo().Pin();
        ELSIF (_inspector.Result = TcoInspectors.eInspectorResult.Passed) THEN
            _inspector.Messenger.Build().Append('I passed').As().AsInfo().Pin();
        END_IF
    END_IF;
END_IF;

END_FUNCTION_BLOCK
